{attribute addProperty BoxType "EL3681-0000-0018"}
{attribute addProperty Id "ControlAT %Q*Control_4BA191DF162"}
{attribute addProperty CRC "2161175933"}
{attribute addProperty SizeInBites "16"}
{attribute addProperty SizeInBytes "2"}
TYPE SAI_Range_80D0ED7D :
STRUCT
	{attribute addProperty Name "Control"}
	Control AT %Q* : Control_4BA191DF;
END_STRUCT
END_TYPE

(* stored: Version 1.2.0.0, ProductVersion 3.1.4024.9
   DUT SAI_Range_80D0ED7D: Id {55f7185c-4827-4867-ba6d-b957039a7f72} *)
